(* IEC 61131-3 sources: RL_MAR/experiments/comparison/llm4plc/results/gpt-4o_20260507_114630/20260507_121247, 1 file *)

(* ---- generated_code_iteration_0.st ---- *)
plaintext
START_ST
FUNCTION_BLOCK FB_FactorialCalculator
VAR_INPUT
    X : INT; // Input variable representing the integer for which the factorial-like values are computed.
END_VAR

VAR_OUTPUT
    FactorialResult : INT; // Output variable representing the final result based on FactorialGoodResult.
    FactorialGoodResult : INT; // Output variable representing X^4.
END_VAR

VAR
    state : INT; // State variable to track the current state of the FSM.
    tempResult : INT; // Temporary variable to hold intermediate calculations during FactorialResult computation.
END_VAR

// Initialization of the state machine
IF state = 0 THEN
    // STATE 0: INITIALIZE
    FactorialGoodResult := 0;
    FactorialResult := 0;
    tempResult := 0;
    state := 1; // Transition to STATE 1 to validate the input range.
END_IF

// Input range validation
IF state = 1 THEN
    // STATE 1: VALIDATE INPUT RANGE
    IF (X >= -3) AND (X <= 3) THEN
        state := 2; // Transition to STATE 2 to compute FactorialGoodResult.
    ELSE
        state := 4; // Transition to STATE 4 to handle out-of-range input.
    END_IF
END_IF

// Compute FactorialGoodResult
IF state = 2 THEN
    // STATE 2: CALCULATE FACTORIALGOODRESULT
    FactorialGoodResult := X * X * X * X; // X^4
    state := 3; // Transition to STATE 3 to compute FactorialResult.
END_IF

// Compute FactorialResult
IF state = 3 THEN
    // STATE 3: CALCULATE FACTORIALRESULT
    IF FactorialGoodResult > 1 THEN
        tempResult := FactorialGoodResult - 1; // Intermediate calculation
        FactorialResult := FactorialGoodResult * tempResult; // FactorialResult = FactorialGoodResult * (FactorialGoodResult - 1)
    ELSE
        FactorialResult := FactorialGoodResult; // FactorialResult = FactorialGoodResult
    END_IF
    state := 0; // Transition back to STATE 0 for the next cycle.
END_IF

// Handle out-of-range input
IF state = 4 THEN
    // STATE 4: HANDLE OUT-OF-RANGE INPUT
    FactorialResult := 1; // Set FactorialResult to 1 to prevent overflow.
    FactorialGoodResult := 0; // FactorialGoodResult is not computed.
    state := 0; // Transition back to STATE 0 for the next cycle.
END_IF

END_FUNCTION_BLOCK
END_ST
